// Mitsubishi GX Works2 project: Step   PLC: Q02U

PROGRAM MAIN
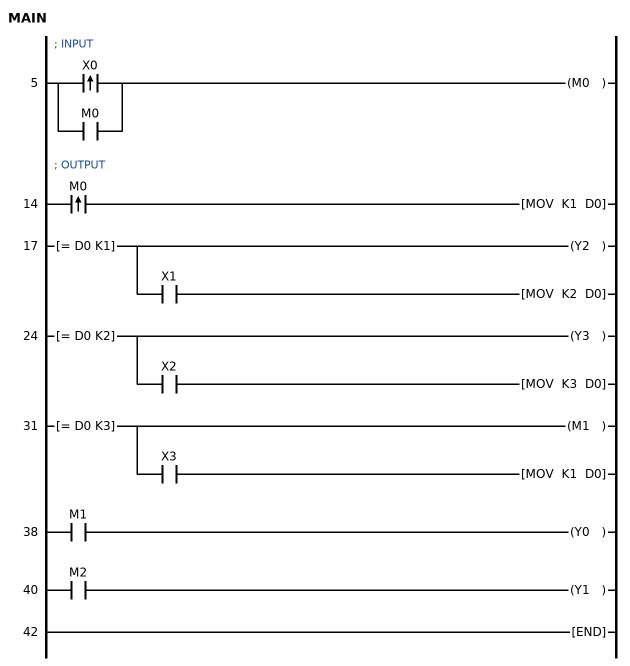
; INPUT
5     LDP     X0
      OR      M0
      OUT     M0
; OUTPUT
14    LDP     M0
      MOV     K1 D0
17    LD=     D0 K1
      OUT     Y2
      AND     X1
      MOV     K2 D0
24    LD=     D0 K2
      OUT     Y3
      AND     X2
      MOV     K3 D0
31    LD=     D0 K3
      OUT     M1
      AND     X3
      MOV     K1 D0
38    LD      M1
      OUT     Y0
40    LD      M2
      OUT     Y1
42    END
END_PROGRAM
